{attribute 'qualified_only'}
{attribute 'strict'}
TYPE E_State :
(
	NormalOperation := 0,
	Simulation		:= 1,
	ConfigMode		:= 2
);
END_TYPE

(* stored: Version 1.1.0.1
   DUT E_State: Id {48a01912-6216-41fa-99d1-49c05e21bff2} *)
